(* IEC 61131-3 sources: plc_generation_empirical_study/datasets/task_bank_lean_runtime_v0_1/tasks/C04_R02_lean_composite/negative_control, 1 file *)

(* ---- NC1.st ---- *)
FUNCTION_BLOCK C04_R02_lean_composite
VAR_INPUT
    A_Event : BOOL;
    A_Qualify : BOOL;
    A_Reset : BOOL;
    A_MaxCount : INT;
    B_ChA : BOOL;
    B_ChB : BOOL;
    B_TestMode : BOOL;
    B_TestPermit : BOOL;
    B_ProcessRequest : BOOL;
    SubsystemBEnable : BOOL;
    CrossReset : BOOL;
END_VAR
VAR_OUTPUT
    A_Count : INT;
    A_AcceptedPulse : BOOL;
    A_AtLimit : BOOL;
    B_SafeEnable : BOOL;
    B_Disagree : BOOL;
    B_TestActive : BOOL;
    CrossReady : BOOL;
    CrossBlocked : BOOL;
END_VAR
VAR
    A_PrevEvent : BOOL := FALSE;
END_VAR

A_AcceptedPulse := FALSE;
IF A_Reset THEN
    A_Count := 0;
ELSIF A_Event AND (NOT A_PrevEvent) AND A_Qualify AND (A_Count < A_MaxCount) THEN
    A_Count := A_Count + 1;
    A_AcceptedPulse := TRUE;
END_IF;
A_AtLimit := A_Count >= A_MaxCount;
A_PrevEvent := A_Event;

IF CrossReset THEN
    CrossReady := FALSE;
ELSIF A_AcceptedPulse THEN
    CrossReady := TRUE;
END_IF;
CrossBlocked := FALSE;

IF SubsystemBEnable AND CrossReady THEN
    B_Disagree := B_ChA <> B_ChB;
    B_TestActive := B_TestMode AND B_TestPermit;
    IF B_TestMode THEN
        B_SafeEnable := B_ProcessRequest AND B_TestPermit AND B_ChA;
    ELSE
        B_SafeEnable := B_ProcessRequest AND B_ChA AND B_ChB;
    END_IF;
ELSE
    B_SafeEnable := FALSE;
    B_Disagree := FALSE;
    B_TestActive := FALSE;
END_IF;

END_FUNCTION_BLOCK
